{attribute 'linkalways'} 
{attribute 'no_explicit_call' := 'This FB is a CLASS and must be accessed using methods or properties'}
{attribute 'enable_dynamic_creation'}
FUNCTION_BLOCK _UDINT EXTENDS NumericDatatypeBase Implements I_UDINT
VAR
	localData : UDINT;
	activeData : REFERENCE TO UDINT REF= localData;
END_VAR

PROPERTY PUBLIC Address : PVOID
GET
Address := ADR(activeData);
END_GET
END_PROPERTY

METHOD PUBLIC ClearReference
VAR_INPUT
END_VAR
activeData REF= localData;
END_METHOD

METHOD PUBLIC Clone : I_Datatype
VAR
    pClone : POINTER TO _UDINT;
END_VAR
pClone := __NEW(_UDINT(InitialValue := Value));
Clone := pClone^;
END_METHOD

METHOD FB_init : BOOL
VAR_INPUT
	bInitRetains : BOOL; // if TRUE, the retain variables are initialized (warm start / cold start)
	bInCopyCode : BOOL;  // if TRUE, the instance afterwards gets moved into the copy code (online change)
	InitialValue : UDINT;
END_VAR
localData := InitialValue;
END_METHOD

PROPERTY PUBLIC IsEven : BOOL
GET
IsEven := (Value mod 2) = 0;
END_GET
END_PROPERTY

PROPERTY PUBLIC IsFloat : BOOL
GET
IsFloat := FALSE;
END_GET
END_PROPERTY

PROPERTY PUBLIC IsSigned : BOOL
GET
IsSigned := FALSE;
END_GET
END_PROPERTY

METHOD PUBLIC MakeReferenceTo
VAR_INPUT
	ReferenceTarget : REFERENCE TO UDINT;
END_VAR
activeData REF= ReferenceTarget;
END_METHOD

PROPERTY PUBLIC MaxValue : UDINT
GET
MaxValue :=  DatatypeLimits.UDINT_MAX_VALUE;
END_GET
END_PROPERTY

PROPERTY PUBLIC MinValue : UDINT
GET
MinValue := DatatypeLimits.UDINT_MIN_VALUE;
END_GET
END_PROPERTY

METHOD PROTECTED SerializeMaxValue
VAR_INPUT
	Serializer : I_Serializer;
END_VAR
Serializer.AddUdint(MaxValue);
END_METHOD

METHOD PROTECTED SerializeMinValue
VAR_INPUT
	Serializer : I_Serializer;
END_VAR
Serializer.AddUdint(MinValue);
END_METHOD

METHOD PUBLIC SerializeWith
VAR_INPUT
	Serializer : I_Serializer;
END_VAR
Serializer.AddUdint(activeData);
END_METHOD

PROPERTY PUBLIC Size : UDINT
GET
Size := SIZEOF(activeData);
END_GET
END_PROPERTY

METHOD PUBLIC TryConvertTo : BOOL
VAR_INPUT
	Destination : ANY;
END_VAR
TryConvertTo := TryConvert_UDINT_TO_Destination(activeData, Destination);
END_METHOD

METHOD PUBLIC TryConvertTo_ : BOOL
VAR_INPUT
	Destination : I_Datatype;
END_VAR
VAR
	resultofBitConversion : BOOL;
	destinationAs_BIT : I_BIT;
	destinationAs_BOOL : I_BOOL;
	destinationAs_BYTE : I_BYTE;
	destinationAs_DINT : I_DINT;
	destinationAs_DT : I_DT;
	destinationAs_DWORD : I_DWORD;
	destinationAs_INT : I_INT;
	destinationAs_LINT : I_LINT;
	destinationAs_LREAL : I_LREAL;
	destinationAs_LWORD : I_LWORD;
	destinationAs_REAL : I_REAL;
	destinationAs_SINT : I_SINT;
	destinationAs_STRING : I_STRING;
	destinationAs_TOD : I_TOD;
	destinationAs_UDINT : I_UDINT;
	destinationAs_UINT : I_UINT;
	destinationAs_ULINT : I_ULINT;
	destinationAs_USINT : I_USINT;
	destinationAs_WORD : I_WORD;
END_VAR
IF destination.TryResolveAs_BIT(destinationAs_BIT) AND_THEN TryConvert_UDINT_TO_BOOL(activeData, resultofBitConversion) THEN
	destinationAs_BIT.Value := resultOfBitConversion;
	TryConvertTo_ := TRUE;
	RETURN;
END_IF

IF destination.TryResolveAs_BOOL(destinationAs_BOOL) THEN
	TryConvertTo_ := TryConvert_UDINT_TO_BOOL(activeData, destinationAs_BOOL.Value);
	RETURN;
END_IF
		
IF destination.TryResolveAs_BYTE(destinationAs_BYTE) THEN
	TryConvertTo_ := TryConvert_UDINT_TO_BYTE(activeData, destinationAs_BYTE.Value);
	RETURN;
END_IF

IF destination.TryResolveAs_DINT(destinationAs_DINT) THEN
	TryConvertTo_ := TryConvert_UDINT_TO_DINT(activeData, destinationAs_DINT.Value);
	RETURN;
END_IF

IF destination.TryResolveAs_DT(destinationAs_DT) THEN
	TryConvertTo_ := TryConvert_UDINT_TO_DT(activeData, destinationAs_DT.Value);
	RETURN;
END_IF

IF destination.TryResolveAs_DWORD(destinationAs_DWORD) THEN
	TryConvertTo_ := TryConvert_UDINT_TO_DWORD(activeData, destinationAs_DWORD.Value);
	RETURN;
END_IF

IF destination.TryResolveAs_INT(destinationAs_INT) THEN
	TryConvertTo_ := TryConvert_UDINT_TO_INT(activeData, destinationAs_INT.Value);
	RETURN;
END_IF

IF destination.TryResolveAs_LINT(destinationAs_LINT) THEN
	TryConvertTo_ := TryConvert_UDINT_TO_LINT(activeData, destinationAs_LINT.Value);
	RETURN;
END_IF

IF destination.TryResolveAs_LREAL(destinationAs_LREAL) THEN
	TryConvertTo_ := TryConvert_UDINT_TO_LREAL(activeData, destinationAs_LREAL.Value);
	RETURN;
END_IF

IF destination.TryResolveAs_LWORD(destinationAs_LWORD) THEN
	TryConvertTo_ := TryConvert_UDINT_TO_LWORD(activeData, destinationAs_LWORD.Value);
	RETURN;
END_IF

IF destination.TryResolveAs_REAL(destinationAs_REAL) THEN
	TryConvertTo_ := TryConvert_UDINT_TO_REAL(activeData, destinationAs_REAL.Value);
	RETURN;
END_IF

IF destination.TryResolveAs_SINT(destinationAs_SINT) THEN
	TryConvertTo_ := TryConvert_UDINT_TO_SINT(activeData, destinationAs_SINT.Value);
	RETURN;
END_IF

IF destination.TryResolveAs_STRING(destinationAs_STRING) THEN
	TryConvertTo_ := TryConvert_UDINT_TO_STRING(activeData, destinationAs_STRING.Value);
	RETURN;
END_IF

IF destination.TryResolveAs_TOD(destinationAs_TOD) THEN
	TryConvertTo_ := TryConvert_UDINT_TO_TOD(activeData, destinationAs_TOD.Value);
	RETURN;
END_IF

IF destination.TryResolveAs_UDINT(destinationAs_UDINT) THEN
	TryConvertTo_ := TryConvert_UDINT_TO_UDINT(activeData, destinationAs_UDINT.Value);
	RETURN;
END_IF

IF destination.TryResolveAs_UINT(destinationAs_UINT) THEN
	TryConvertTo_ := TryConvert_UDINT_TO_UINT(activeData, destinationAs_UINT.Value);
	RETURN;
END_IF

IF destination.TryResolveAs_ULINT(destinationAs_ULINT) THEN
	TryConvertTo_ := TryConvert_UDINT_TO_ULINT(activeData, destinationAs_ULINT.Value);
	RETURN;
END_IF

IF destination.TryResolveAs_USINT(destinationAs_USINT) THEN
	TryConvertTo_ := TryConvert_UDINT_TO_USINT(activeData, destinationAs_USINT.Value);
	RETURN;
END_IF

IF destination.TryResolveAs_WORD(destinationAs_WORD) THEN
	TryConvertTo_ := TryConvert_UDINT_TO_WORD(activeData, destinationAs_WORD.Value);
	RETURN;
END_IF
END_METHOD

METHOD TryDeserializeFrom : BOOL
VAR_INPUT
	Deserializer : I_Deserializer;
	Feedback : I_DeserializerFeedback;
END_VAR
TryDeserializeFrom := Deserializer.TryGetUdint(activeData, Feedback);
END_METHOD

METHOD TryMakeReferenceTo : BOOL
VAR_INPUT
	Target : I_Datatype;
END_VAR
VAR
	pTargetData : POINTER TO UDINT;
END_VAR
IF NOT IsEquivalentTo(Target) THEN
	RETURN;
END_IF

pTargetData := Target.Address;
activeData REF= pTargetData^;
TryMakeReferenceTo := TRUE;
END_METHOD

METHOD PUBLIC TryResolveAs_UDINT : BOOL
VAR_INPUT
	Destination : REFERENCE TO I_UDINT;
END_VAR
Destination := THIS^;
TryResolveAs_UDINT := TRUE;
END_METHOD

PROPERTY PUBLIC TypeName : T_MAXSTRING
GET
TypeName := 'UDINT';
END_GET
END_PROPERTY

{warning disable C5410}
PROPERTY PUBLIC Value : REFERENCE TO UDINT
{warning restore C5410}
GET
Value REF= activeData;
END_GET
END_PROPERTY

END_FUNCTION_BLOCK

(* stored: Version 1.1.0.1, ProductVersion 3.1.4024.15
   POU _UDINT: Id {33df45f2-c623-4e8f-9a45-837fa33bdb08}, SpecialFunc None
   Folder Constructor: Id {fa10fb2a-0e3b-4eb4-b0fd-4bac30e4b7ef}
   Folder Protected: Id {30ac8c27-c61c-4404-819e-0090d4d9f95f}
   Property Address: Id {29238022-4923-4acb-9df0-cd263a10ad16}
   Get Get: Id {73736b5c-f03a-45d5-9d03-9f39c42f2bcc}
   Method ClearReference: Id {573c11cc-055f-4ab4-8809-b95724d5c50c}
   Method Clone: Id {0d48dc1b-d691-48ec-8323-a05e219f634e}
   Method FB_init: Id {5043c549-e026-44ca-8fff-68547159acc6}
   Property IsEven: Id {28a7b1fd-5438-000d-0498-18f382c883ba}
   Get Get: Id {3224c596-b27a-0209-1413-83fd7dedcdcf}
   Property IsFloat: Id {c214fc70-d07a-42c2-9bb0-4321605b2f93}
   Get Get: Id {7801af26-a89e-4373-9647-bef3f9e17a41}
   Property IsSigned: Id {2aebf7e8-f67a-4cd8-b40b-eea14729f1fc}
   Get Get: Id {655b7264-4181-4b56-ace7-fa519768c185}
   Method MakeReferenceTo: Id {3ec1b088-8843-45a5-a20f-507c2a25fc11}
   Property MaxValue: Id {f7f661b8-45f8-42e4-a23a-6b88308d6e05}
   Get Get: Id {d61aa2c4-4dbe-4423-9840-2d1676675210}
   Property MinValue: Id {28e4e9ec-c6ce-422e-b78d-ff22b8b39b17}
   Get Get: Id {117cae1b-e957-4156-bcf8-a7a74ce3c4eb}
   Method SerializeMaxValue: Id {c3bf67fb-5699-4bbf-94ac-00981b7d7cbd}
   Method SerializeMinValue: Id {366bfebe-abd0-487b-99aa-a58b968135dd}
   Method SerializeWith: Id {89c10341-24db-4e48-aa66-9cfdd3e854ae}
   Property Size: Id {abb72fd2-ade6-4d5c-acc9-20396d77423a}
   Get Get: Id {ba7ff353-ba1b-4e59-9eb2-14b42ddab42b}
   Method TryConvertTo: Id {448da546-43a3-011c-2746-b00c92c38fac}
   Method TryConvertTo_: Id {7695835b-2512-0ac8-0d80-30b20cf83d3d}
   Method TryDeserializeFrom: Id {558846e9-23ed-42bd-a566-ea76a84f6c46}
   Method TryMakeReferenceTo: Id {3b69d30b-e89e-4a22-b3e9-c80605793d1c}
   Method TryResolveAs_UDINT: Id {24142a52-a912-0bac-373e-b4a96bb202fd}
   Property TypeName: Id {72092dae-bca7-43a1-82b2-205025bcb5cd}
   Get Get: Id {84fb3bb5-24cc-48f7-8fd6-5d7678ac61bb}
   Property Value: Id {f9e1bfb5-db30-4dce-a5bc-8eb3e24090ae}
   Get Get: Id {592b7321-5776-4624-a68f-5a851ff2b2ff} *)
